// TIA Portal V21 export
ORGANIZATION_BLOCK "Startup"   // OB100, LAD, Startup
TITLE = "Complete Restart"
{ S7_Optimized_Access := 'TRUE' }
// stored: AutoNumber false, SetENOAutomatically false
   VAR_INPUT
      LostRetentive : Bool;   // True if retentive data are lost
      LostRTC : Bool;   // True if date and time are lost
   END_VAR
BEGIN

REGION Network 1
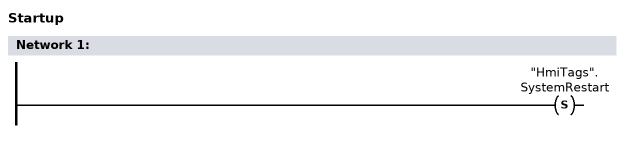
   RUNG wire#powerrail
      S_Coil( "HmiTags".SystemRestart )
   END_RUNG
   // the same network as SCL:
   "HmiTags".SystemRestart := TRUE;
END_REGION
END_ORGANIZATION_BLOCK
